{attribute 'GeneratedUsingTerminal: EP1859-0042-0019'}
{attribute addProperty BoxType "EP1859-0042-0019"}
{attribute addProperty Id "OutputAT %Q*BOOL1"}
{attribute addProperty CRC "1120571895"}
{attribute addProperty Size "1"}
TYPE DO_X_42CA91F7 :
STRUCT
	{attribute addProperty Name "Output"}
	Output AT %Q* : BOOL;
END_STRUCT
END_TYPE

(* stored: Version 1.2.0.0, ProductVersion 3.1.4024.9
   DUT DO_X_42CA91F7: Id {65ba3e4a-33ee-42bd-a303-8750a4106f51} *)
